FUNCTION_BLOCK FB_Bank
VAR_INPUT
	sBankName : STRING(200);
END_VAR

VAR
	fBalance : REAL;
END_VAR

fMoney := 4343;

{attribute 'monitoring' := 'call'}
PROPERTY PROTECTED fMoney : REAL
GET
fMoney := fBalance;
END_GET
SET // PRIVATE
fBalance := fMoney;
END_SET
END_PROPERTY

METHOD M_Deposit : BOOL
VAR_INPUT
	fDepositAmount : REAL;
END_VAR
fMoney := fDepositAmount;
END_METHOD

METHOD M_Withdrawal : BOOL
VAR_INPUT
	fWithdrawAmount : REAL;
END_VAR
IF fWithdrawAmount <= fMoney THEN
	fMoney := fMoney - fWithdrawAmount;
END_IF
END_METHOD

END_FUNCTION_BLOCK

(* stored: Version 1.1.0.1, ProductVersion 3.1.4024.16
   POU FB_Bank: Id {d56d0523-3941-407a-937d-e5d4e0e4bc5a}, SpecialFunc None
   Property fMoney: Id {8824347c-e9d9-4936-bdea-922df011b715}
   Get Get: Id {238ef373-05c3-4513-85ef-0a7bc5990195}
   Set Set: Id {b43ef411-2265-4a32-ac55-79f27981fea8}
   Method M_Deposit: Id {43d1d39d-abc9-4455-a6e4-11b4165b22a6}
   Method M_Withdrawal: Id {c4e7d9f3-0a54-4fe8-adb5-dad00b7a3b92} *)
